INTERFACE I_ExternalSetpointGenerator


METHOD Disable
VAR_OUTPUT
    Done : BOOL;
    Busy : BOOL;
    Error : BOOL;
    ErrorID : UDINT;
    Enabled : BOOL;
END_VAR
END_METHOD

PROPERTY DisableBusy : BOOL
GET
END_GET
END_PROPERTY

PROPERTY DisableDone : BOOL
GET
END_GET
END_PROPERTY


METHOD Enable
VAR_OUTPUT
    Done : BOOL;
    Busy : BOOL;
    Error : BOOL;
    ErrorID : UDINT;
    Enabled : BOOL;
END_VAR
END_METHOD

PROPERTY EnableBusy : BOOL
GET
END_GET
END_PROPERTY

PROPERTY EnableDone : BOOL
GET
END_GET
END_PROPERTY

PROPERTY EnableError : BOOL
GET
END_GET
END_PROPERTY


METHOD Halt
VAR_OUTPUT
    Done : BOOL;
    Busy : BOOL;
    Active : BOOL;
    CommandAborted : BOOL;
    Error : BOOL;
    ErrorID : UDINT;
END_VAR
END_METHOD

PROPERTY HaltBusy : BOOL
GET
END_GET
END_PROPERTY

PROPERTY HaltDone : BOOL
GET
END_GET
END_PROPERTY


METHOD IsEnabled : BOOL
END_METHOD


METHOD SetAcceleraSetpoint
VAR_INPUT
    Setpoint : LREAL;
END_VAR
VAR_OUTPUT
	Error : BOOL;
	ErrorMsg : T_MaxString;
END_VAR
END_METHOD


METHOD SetPositionSetpoint
VAR_INPUT
    Setpoint : LREAL;
END_VAR
VAR_OUTPUT
	Error : BOOL;
	ErrorMsg : T_MaxString;
END_VAR
END_METHOD


METHOD SetSetpoints
VAR_INPUT
    PositionSetpoint : LREAL;
    VelocitySetpoint : LREAL;
    AcceleraSetpoint : LREAL;
END_VAR
VAR_OUTPUT
	Error : BOOL;
	ErrorMsg : T_MaxString;
END_VAR
END_METHOD


METHOD SetVelocitySetpoint
VAR_INPUT
    Setpoint : LREAL;
END_VAR
VAR_OUTPUT
	Error : BOOL;
	ErrorMsg : T_MaxString;
END_VAR
END_METHOD

END_INTERFACE

(* stored: Version 1.1.0.1
   Itf I_ExternalSetpointGenerator: Id {256ff4ab-16a6-4272-805e-f8c2c4343ca7}
   Method Disable: Id {1f93fc3c-1418-47fc-ac86-a566b1fee5ff}
   Property DisableBusy: Id {9fb201ef-e8a1-4ec5-88ca-604c23f88aa2}
   Get Get: Id {2a6d1d0d-f6a2-44bf-9775-1fe73ccecf74}
   Property DisableDone: Id {fc5e48ee-b3a8-4bff-a257-64f175da12fc}
   Get Get: Id {a4a35d4f-1aec-4e8e-a296-eefaec70efdb}
   Method Enable: Id {5879e138-2b2e-4380-8b6f-7002c85d15b0}
   Property EnableBusy: Id {0decd41e-537f-4cfd-8d69-e42d83825ef9}
   Get Get: Id {4630aa56-3cd3-44fb-b693-9fca8f02191b}
   Property EnableDone: Id {929f91bd-806b-4bad-9fe1-43e79d9f9645}
   Get Get: Id {a5a72456-1883-4324-b8f5-9b823fa32a1b}
   Property EnableError: Id {c9799f06-8fb5-4bf9-abe4-13cc65439287}
   Get Get: Id {8f92eae8-ac82-497b-8369-a096f348a007}
   Method Halt: Id {84ade41b-2dca-4d65-a351-2bb3a51aefb4}
   Property HaltBusy: Id {020b31a1-469d-48cb-920b-684056a0f9fa}
   Get Get: Id {24a606bc-d706-4870-90d6-1ed182880c09}
   Property HaltDone: Id {7321c2cb-3723-4833-8fa7-0f267407315b}
   Get Get: Id {a5411a2b-9662-4b7f-bdf4-c3ee078c1ca5}
   Method IsEnabled: Id {cf2be58d-de83-47be-9f57-f4460ca6763f}
   Method SetAcceleraSetpoint: Id {4ebad5ae-3852-4642-8c9b-5e716adcfad0}
   Method SetPositionSetpoint: Id {f7ebbd29-ed8b-479e-ad3e-974d575d8bcf}
   Method SetSetpoints: Id {5ba30d0b-50f3-40c9-8cff-d9ede3d0f1e0}
   Method SetVelocitySetpoint: Id {2e9418d5-d761-41de-8a6f-f12b0c8e9919} *)
